FUNCTION ATAN2_deg : LREAL
VAR_INPUT	
    y : REAL; // y-coordinate
    x : REAL; // x-coordinate
END_VAR
VAR_OUTPUT
END_VAR

IF x > 0 THEN
    ATAN2_deg := ATAN(y / x);
ELSIF x < 0 AND y >= 0 THEN
    ATAN2_deg := ATAN(y / x) + pi;
ELSIF x < 0 AND y < 0 THEN
    ATAN2_deg := ATAN(y / x) - pi;
ELSIF x = 0 AND y > 0 THEN
    ATAN2_deg := pi / 2;
ELSIF x = 0 AND y < 0 THEN
    ATAN2_deg := -pi / 2;
ELSIF x = 0 AND y = 0 THEN
    ATAN2_deg := 0.0; // Undefined, but conventionally set to 0
END_IF

END_FUNCTION

(* stored: Version 1.1.0.1, ProductVersion 3.1.4024.13
   POU ATAN2_deg: Id {b0d4148c-2f7d-449c-ab08-e08d9f539b26}, SpecialFunc None *)
